FUNCTION_BLOCK CompositeBlock
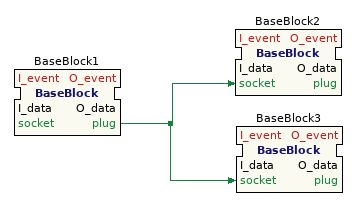
  FBS
    BaseBlock1 : BaseBlock;
    BaseBlock2 : BaseBlock;
    BaseBlock3 : BaseBlock;
  END_FBS
  ADAPTER_CONNECTIONS
    BaseBlock1.plug TO BaseBlock2.socket;
    BaseBlock1.plug TO BaseBlock3.socket;
  END_CONNECTIONS
END_FUNCTION_BLOCK
